// TIA Portal V14 export
FUNCTION_BLOCK "FB_MotorControl"   // FB1, SCL
// stored: AutoNumber true
BEGIN
END_FUNCTION_BLOCK
